FUNCTION FC10_Alias : BOOL
VAR_INPUT
END_VAR
VAR
END_VAR

// IO vertaling van tag naar in en uitgangen
// schalen van analoge ingangen naar tagwaarden en andersom

// als we analoge spul hebben lol

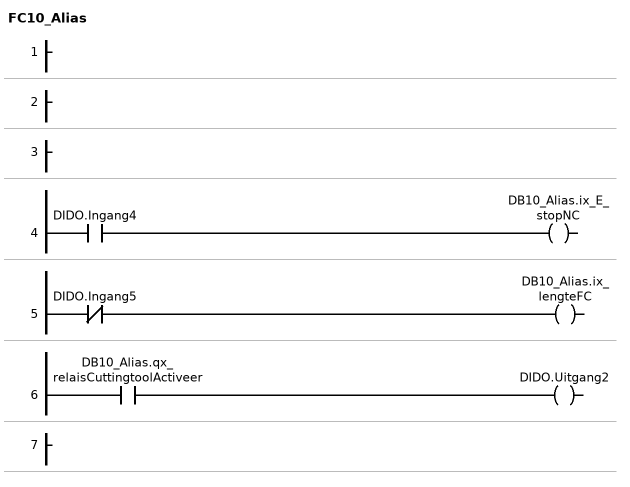
// NETWORK 1

// NETWORK 2

// NETWORK 3

// NETWORK 4
DB10_Alias.ix_E_stopNC := DIDO.Ingang4;

// NETWORK 5
DB10_Alias.ix_lengteFC := NOT DIDO.Ingang5;

// NETWORK 6
DIDO.Uitgang2 := DB10_Alias.qx_relaisCuttingtoolActiveer;

// NETWORK 7

END_FUNCTION

(* stored: Version 1.1.0.1, ProductVersion 3.1.4024.12
   POU FC10_Alias: Id {b9e40a38-81b0-4072-8db3-c7add526f050}, SpecialFunc None *)
